PROGRAM PRG_SafetyHandle
VAR
	//Air Supply testing
	bAirSupplyEnable: BOOL	:= TRUE;
	bAirSupplyReset	: BOOL	:= FALSE;
	
	bLockDoors	  	: BOOL 	:= FALSE;	   	// Variable that sends the lock doors signal
	
	tonStabilizingFaults : TON;
	tonClearFaults		 : TON;
	
	i	: USINT;
END_VAR

//Safety Restart & Error Ack
IF GVL_Safety.SafetyInputs.bMachineReset OR GVL_Safety.bM1STOErrorAck THEN
	GVL_Safety.bSafetyErrorAck			:= TRUE;
	GVL_Motion.M1Motor.bTS_ErrorAck		:= TRUE;
ELSE
	GVL_Safety.bSafetyErrorAck			:= FALSE;
	GVL_Motion.M1Motor.bTS_ErrorAck		:= FALSE;
END_IF

GVL_Safety.iM4STOErrorAck			:= GVL_Safety.SafetyInputs.bMachineReset;
GVL_Safety.iM5STOErrorAck			:= GVL_Safety.SafetyInputs.bMachineReset;
GVL_Safety.iM6STOErrorAck			:= GVL_Safety.SafetyInputs.bMachineReset;
GVL_Safety.iM7STOErrorAck			:= GVL_Safety.SafetyInputs.bMachineReset;
GVL_Safety.iM8STOErrorAck			:= GVL_Safety.SafetyInputs.bMachineReset;

GVL_Safety.bSafetyRun				:= TRUE;
GVL_Motion.M1Motor.bTS_Run			:= TRUE;
GVL_Safety.iM4STORun				:= TRUE;
GVL_Safety.iM5STORun				:= TRUE;
GVL_Safety.iM6STORun				:= TRUE;
GVL_Safety.iM7STORun				:= TRUE;
GVL_Safety.iM8STORun				:= TRUE;

IF bAirSupplyEnable THEN
	GVL_Safety.bAirSupplyEnable := TRUE;
ELSE
	GVL_Safety.bAirSupplyEnable	:= FALSE;
END_IF

IF bAirSupplyReset THEN
	GVL_Safety.bAirSupplyReset 	:= TRUE;
ELSE
	GVL_Safety.bAirSupplyReset	:= FALSE;
END_IF

//Alias signal for the reset button blinking
IF GVL_Safety.bResetButtonBlink THEN
	GVL_IO.gDigOutputs.bResetIndicator	:= TRUE;
ELSE
	GVL_IO.gDigOutputs.bResetIndicator	:= FALSE;
END_IF

IF bLockDoors THEN
	GVL_Safety.SafetyOutputs.bLockDoorSafety := TRUE;
	ELSE
	GVL_Safety.SafetyOutputs.bLockDoorSafety := FALSE;
END_IF

// ====================================================================
// 1. SAFETY FAULT LOGIC (STOP & DISABLE ALL PUMPS)
// ====================================================================
// This section executes every PLC cycle while the safety condition is NOT met.

IF NOT GVL_Safety.bSafetyEnable AND GVL_Motion.bInitialHomingDone THEN
	// Immediate Stop and Disable all pumps and linear motors for safety
	FOR i := 1 TO 10 DO
		// 1. Initiate Controlled Stop (MC_Stop) to cancel any active motion commands
		GVL_Motion.aPumpsRotary[i].Stop(); 
		GVL_Motion.aPumpsLinear[i].Stop();
		
		// 2. Immediate Torque Cut-Off (MC_Power.Enable := FALSE)
		GVL_Motion.aPumpsRotary[i].Disable();
		GVL_Motion.aPumpsLinear[i].Disable();
	END_FOR
END_IF

// ====================================================================
// 2. Immediate Fault Command from software conditions
// ====================================================================
// This section activates an immediate fault from alarms flags 

IF GVL_Safety.bSafetyEnable THEN
	GVL_Safety.bImmediateFaultCommand := 
	GVL_Alarms.arrEventFlag[50] OR GVL_Alarms.arrEventFlag[51] OR GVL_Alarms.arrEventFlag[52] OR 
	GVL_Alarms.arrEventFlag[53] OR GVL_Alarms.arrEventFlag[54] OR GVL_Alarms.arrEventFlag[55] OR 
	GVL_Alarms.arrEventFlag[56] OR GVL_Alarms.arrEventFlag[57] OR GVL_Alarms.arrEventFlag[58] OR 
	GVL_Alarms.arrEventFlag[59] OR GVL_Alarms.arrEventFlag[60] OR GVL_Alarms.arrEventFlag[61] OR 
	GVL_Alarms.arrEventFlag[62] OR GVL_Alarms.arrEventFlag[63] OR GVL_Alarms.arrEventFlag[64] OR 
	GVL_Alarms.arrEventFlag[65] OR GVL_Alarms.arrEventFlag[66] OR GVL_Alarms.arrEventFlag[67] OR 
	GVL_Alarms.arrEventFlag[68] OR GVL_Alarms.arrEventFlag[69] OR GVL_Alarms.arrEventFlag[70] OR 
	GVL_Alarms.arrEventFlag[71] OR GVL_Alarms.arrEventFlag[72] OR GVL_Alarms.arrEventFlag[73] OR 
	GVL_Alarms.arrEventFlag[74] OR GVL_Alarms.arrEventFlag[75] OR GVL_Alarms.arrEventFlag[76] OR 
	GVL_Alarms.arrEventFlag[77] OR GVL_Alarms.arrEventFlag[78] OR GVL_Alarms.arrEventFlag[79] OR 
	GVL_Alarms.arrEventFlag[80] OR GVL_Alarms.arrEventFlag[81] OR GVL_Alarms.arrEventFlag[82] OR 
	GVL_Alarms.arrEventFlag[83] OR GVL_Alarms.arrEventFlag[84] OR GVL_Alarms.arrEventFlag[85] OR 
	GVL_Alarms.arrEventFlag[86] OR GVL_Alarms.arrEventFlag[200] OR GVL_Alarms.arrEventFlag[201] OR
	GVL_Alarms.arrEventFlag[202] OR GVL_Alarms.arrEventFlag[203] OR (*GVL_Alarms.arrEventFlag[204] OR*) 
	GVL_Alarms.arrEventFlag[205] OR GVL_Alarms.arrEventFlag[206] OR GVL_Alarms.arrEventFlag[207] OR 
	GVL_Alarms.arrEventFlag[208] OR GVL_Alarms.arrEventFlag[209] OR GVL_Alarms.arrEventFlag[210] OR 
	GVL_Alarms.arrEventFlag[211] OR GVL_Alarms.arrEventFlag[212] OR GVL_Alarms.arrEventFlag[213] OR 
	GVL_Alarms.arrEventFlag[214] OR GVL_Alarms.arrEventFlag[215] OR GVL_Alarms.arrEventFlag[216] OR 
	GVL_Alarms.arrEventFlag[217] OR GVL_Alarms.arrEventFlag[218] OR GVL_Alarms.arrEventFlag[219] OR 
	GVL_Alarms.arrEventFlag[220] OR GVL_Alarms.arrEventFlag[221] OR GVL_Alarms.arrEventFlag[222] OR 
	GVL_Alarms.arrEventFlag[223] OR GVL_Alarms.arrEventFlag[224];
ELSE
	GVL_Safety.bImmediateFaultCommand := FALSE;
END_IF

END_PROGRAM

(* stored: Version 1.1.0.1, ProductVersion 3.1.4024.15
   POU PRG_SafetyHandle: Id {8e15bf43-686d-46b2-be47-568f063f8b7c}, SpecialFunc None *)
